FUNCTION F_LeakMonitor_LOTNL_1 : FB_LeakMonitor
VAR_INPUT
END_VAR
VAR_OUTPUT
	// Provide stBoundaries output so test functions can reuse the boundaries
	stBoundaries : ST_LeakBoundaries := F_LeakBoundaries();
END_VAR
VAR
	fbLeakMonitor : FB_LeakMonitor;
END_VAR

fbLeakMonitor(
	bLeakDetected := TRUE,
	nLocationResistance := stBoundaries.nLMax4 - 1,
	stBound := stBoundaries,
);

F_LeakMonitor_LOTNL_1 := fbLeakMonitor;

END_FUNCTION

(* stored: Version 1.1.0.1, ProductVersion 3.1.4024.0
   POU F_LeakMonitor_LOTNL_1: Id {c9f0ccb7-aeed-4622-8418-8dd1776bc54e}, SpecialFunc None *)
